(* PLC project balance, Dassault Systèmes ControlBuild 2024x *)
(* stored: creationDateTime 2023-10-03T11:12:58-01:00 *)

(* This module simulates the behaviour of a balance with calibration and reset of weight. *)
FUNCTION_BLOCK equipment_library.balance
  VAR_INPUT
    reset : BOOL := false;
    weight : REAL := 0.0;
    calibration : BOOL := false;
  END_VAR
  VAR_OUTPUT
    valueWeight : REAL := 0.0;
    stableWeight : BOOL := false;
  END_VAR
  VAR
    tare : REAL := 0.0;
    oldWeight : REAL := 0.0;
  END_VAR
  VAR CONSTANT
    stableLogic : BOOL := true;
  END_VAR
  VAR
    d_stable : BOOL := false;
    v_d_stable : BOOL := false;
    d_measure : BOOL := false;
    v_d_measure : REAL := 0.0;
  END_VAR


ACTION C_source_code:
/* -----------------------------------------------------------------	*/
/* Type : Model of Operative Behaviour					*/
/* Catégorie :   batch							*/
/* Author : Dassault Systemes						*/
/* Update date : June 2018							*/
/* -----------------------------------------------------------------	*/
/* This module simulates the behaviour of a balance with zero point	*/
/* adjustment and reset of weight.						*/
/* If the weight is stable, the command task can use the weigth.	*/
/* ----------------------------------------------------------------- */


/* ----------------------------------------------------------------	*/
/* Calibration adjusting				 			*/
/* ----------------------------------------------------------------	*/
if(FM(calibration))  tare=weight;

/* ----------------------------------------------------------------	*/
/* Computing of weight 							*/
/* ----------------------------------------------------------------	*/
if (d_measure) valueWeight = v_d_measure;
else valueWeight=weight-tare;

/* ----------------------------------------------------------------	*/
/* Reset of weight 								*/
/* ----------------------------------------------------------------	*/
if((reset)) tare=0;

/* ----------------------------------------------------------------	*/
/* Stability of weight 							*/
/* ----------------------------------------------------------------	*/
if(oldWeight!=weight) stableWeight=!stableLogic;
if(d_stable) stableWeight=v_d_stable^!stableLogic;
oldWeight=weight;
END_ACTION
END_FUNCTION_BLOCK
